// TIA Portal V20 export
// export: Created 2025-12-01T14:56:58.1690783Z, ExportSetting None, DisplayName Totally Integrated Automation Portal, DisplayVersion V20 Update 3, DisplayName TIA Portal Openness, DisplayVersion V20 Update 3, DisplayName TIA Portal Version Control Interface, DisplayVersion V20 Update 3, DisplayName STEP 7 Professional, DisplayVersion V20 Update 3, DisplayName STEP 7 Safety, DisplayVersion V20 Update 2, DisplayName WinCC Basic/Comfort/Advanced, DisplayVersion V20 Update 3, DisplayName WinCC Professional, DisplayVersion V20 Update 3, DisplayName WinCC Unified, DisplayVersion V20 Update 3
FUNCTION_BLOCK "FB86_GALIBO_3Laterales"   // FB86, LAD
TITLE = Galibo de 3 Anchuras (2024)
{ S7_Optimized_Access := 'FALSE' }
AUTHOR : GALIBO
NAME : 20140101
VERSION : 3.0
// stored: AutoNumber false, SetENOAutomatically false
   VAR_INPUT
      Mesa : UInt;
      NumGalibo : UInt;
      EnRodillos : Bool;
      pHs_Lateral_Dcha_Err : Bool;
      pHs_Lateral_Dcha_2 : Bool;
      pHs_Lateral_Dcha_1 : Bool;
      pHs_Lateral_Izq_1 : Bool;
      pHs_Lateral_Izq_2 : Bool;
      pHs_Lateral_Izq_Err : Bool;
      HabilitarLectura : Bool;
      PermisoLectura : Bool;
      Rearmar_ConMesaLibre : Bool;
   END_VAR
   VAR_OUTPUT
      Baliza : Bool;
      ErrorLateral : Bool;
      FinLectura : Bool;
   END_VAR
   VAR
      GAL_ET00 : Bool;
      GAL_ET01 : Bool;
      GAL_ET02 : Bool;
      GAL_ET03 : Bool;
      pHsGalibo_OK { ExternalAccessible := 'False'; ExternalVisible := 'False'; ExternalWritable := 'False'} : Bool;
      Lateral_NOOK_Dcha : Bool;
      Lateral_NOOK_Izq : Bool;
      Lateral_OK_1 : Bool;
      Lateral_OK_2 : Bool;
      Lateral_OK_3 : Bool;
      LeerLateral : Bool;
      CodigoLateral : SInt;
      MemoCodigo : Word;
      STAT_Baliza_Galibo : Bool;
   END_VAR
   VAR_TEMP
      EstadoZona : "EstadoZona";
      EstadoVI : "EstadosMesa";
   END_VAR
   VAR_TEMP   // added for the SCL form of the ladder/FBD networks
      _w1 : Bool;
   END_VAR
BEGIN

REGION Network 1: INICIALIZAR - Recoger las Variables de Estado de la Mesa
   // Se recoge - Estado_CBx
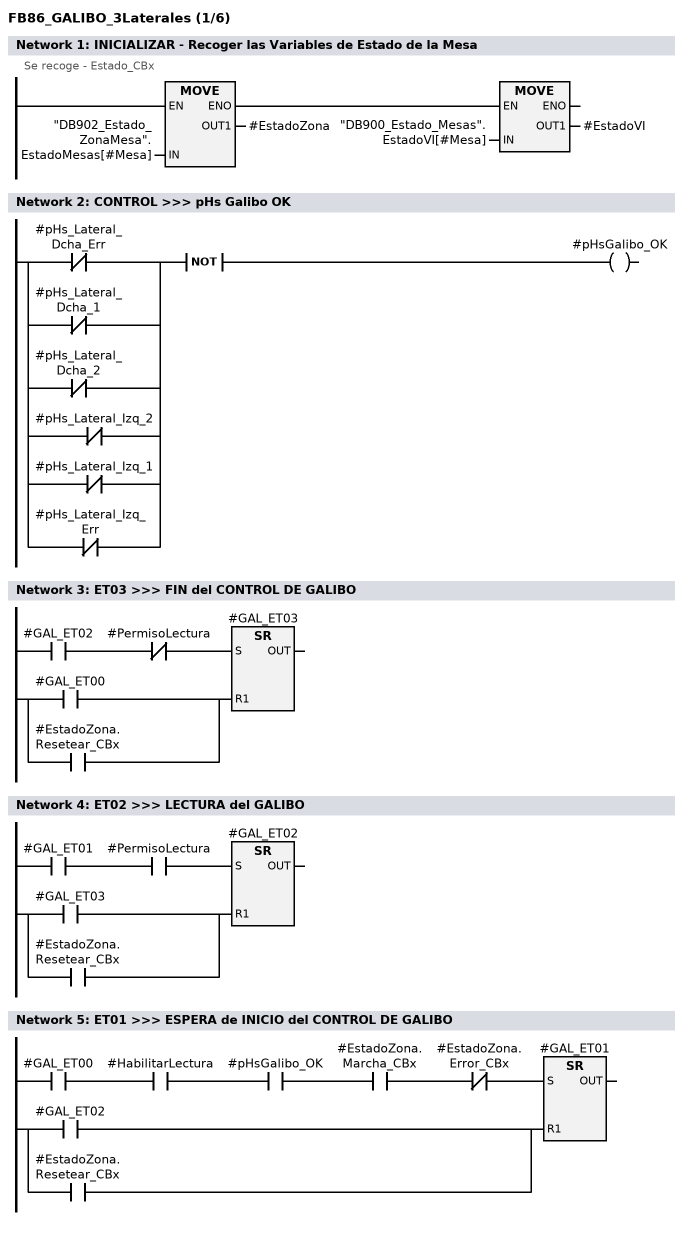
   RUNG wire#powerrail
      Move(in := "DB902_Estado_ZonaMesa".EstadoMesas[#Mesa], out1 => #EstadoZona)
      Move(in := "DB900_Estado_Mesas".EstadoVI[#Mesa], out1 => #EstadoVI)
   END_RUNG
   // the same network as SCL:
   #EstadoZona := "DB902_Estado_ZonaMesa".EstadoMesas[#Mesa];
   #EstadoVI := "DB900_Estado_Mesas".EstadoVI[#Mesa];
END_REGION

REGION Network 2: CONTROL >>> pHs Galibo OK
   RUNG wire#powerrail
      I_Contact( #pHs_Lateral_Dcha_Err )
      wire#w1
      Not()
      Coil( #pHsGalibo_OK )
   END_RUNG
   RUNG wire#powerrail
      I_Contact( #pHs_Lateral_Dcha_1 )
   END_RUNG wire#w1
   RUNG wire#powerrail
      I_Contact( #pHs_Lateral_Dcha_2 )
   END_RUNG wire#w1
   RUNG wire#powerrail
      I_Contact( #pHs_Lateral_Izq_2 )
   END_RUNG wire#w1
   RUNG wire#powerrail
      I_Contact( #pHs_Lateral_Izq_1 )
   END_RUNG wire#w1
   RUNG wire#powerrail
      I_Contact( #pHs_Lateral_Izq_Err )
   END_RUNG wire#w1
   // the same network as SCL:
   #pHsGalibo_OK := NOT (NOT #pHs_Lateral_Dcha_Err OR NOT #pHs_Lateral_Dcha_1 OR NOT #pHs_Lateral_Dcha_2 OR NOT #pHs_Lateral_Izq_2 OR NOT #pHs_Lateral_Izq_1 OR NOT #pHs_Lateral_Izq_Err);
END_REGION

REGION Network 3: ET03 >>> FIN del CONTROL DE GALIBO
   RUNG wire#powerrail
      Contact( #GAL_ET02 )
      I_Contact( #PermisoLectura )
      S_SR(operand := #GAL_ET03, r1 := wire#w1)
   END_RUNG
   RUNG wire#powerrail
      Contact( #GAL_ET00 )
   END_RUNG wire#w1
   RUNG wire#powerrail
      Contact( #EstadoZona.Resetear_CBx )
   END_RUNG wire#w1
   // the same network as SCL:
   IF #GAL_ET02 AND NOT #PermisoLectura THEN
       #GAL_ET03 := TRUE;   // SR flip-flop
   END_IF;
   IF #GAL_ET00 OR #EstadoZona.Resetear_CBx THEN #GAL_ET03 := FALSE; END_IF;
END_REGION

REGION Network 4: ET02 >>> LECTURA del GALIBO
   RUNG wire#powerrail
      Contact( #GAL_ET01 )
      Contact( #PermisoLectura )
      S_SR(operand := #GAL_ET02, r1 := wire#w1)
   END_RUNG
   RUNG wire#powerrail
      Contact( #GAL_ET03 )
   END_RUNG wire#w1
   RUNG wire#powerrail
      Contact( #EstadoZona.Resetear_CBx )
   END_RUNG wire#w1
   // the same network as SCL:
   IF #GAL_ET01 AND #PermisoLectura THEN
       #GAL_ET02 := TRUE;   // SR flip-flop
   END_IF;
   IF #GAL_ET03 OR #EstadoZona.Resetear_CBx THEN #GAL_ET02 := FALSE; END_IF;
END_REGION

REGION Network 5: ET01 >>> ESPERA de INICIO del CONTROL DE GALIBO
   RUNG wire#powerrail
      Contact( #GAL_ET00 )
      Contact( #HabilitarLectura )
      Contact( #pHsGalibo_OK )
      Contact( #EstadoZona.Marcha_CBx )
      I_Contact( #EstadoZona.Error_CBx )
      S_SR(operand := #GAL_ET01, r1 := wire#w1)
   END_RUNG
   RUNG wire#powerrail
      Contact( #GAL_ET02 )
   END_RUNG wire#w1
   RUNG wire#powerrail
      Contact( #EstadoZona.Resetear_CBx )
   END_RUNG wire#w1
   // the same network as SCL:
   IF #GAL_ET00 AND #HabilitarLectura AND #pHsGalibo_OK AND #EstadoZona.Marcha_CBx AND NOT #EstadoZona.Error_CBx THEN
       #GAL_ET01 := TRUE;   // SR flip-flop
   END_IF;
   IF #GAL_ET02 OR #EstadoZona.Resetear_CBx THEN #GAL_ET01 := FALSE; END_IF;
END_REGION

REGION Network 6: ET00 >>> INICIO
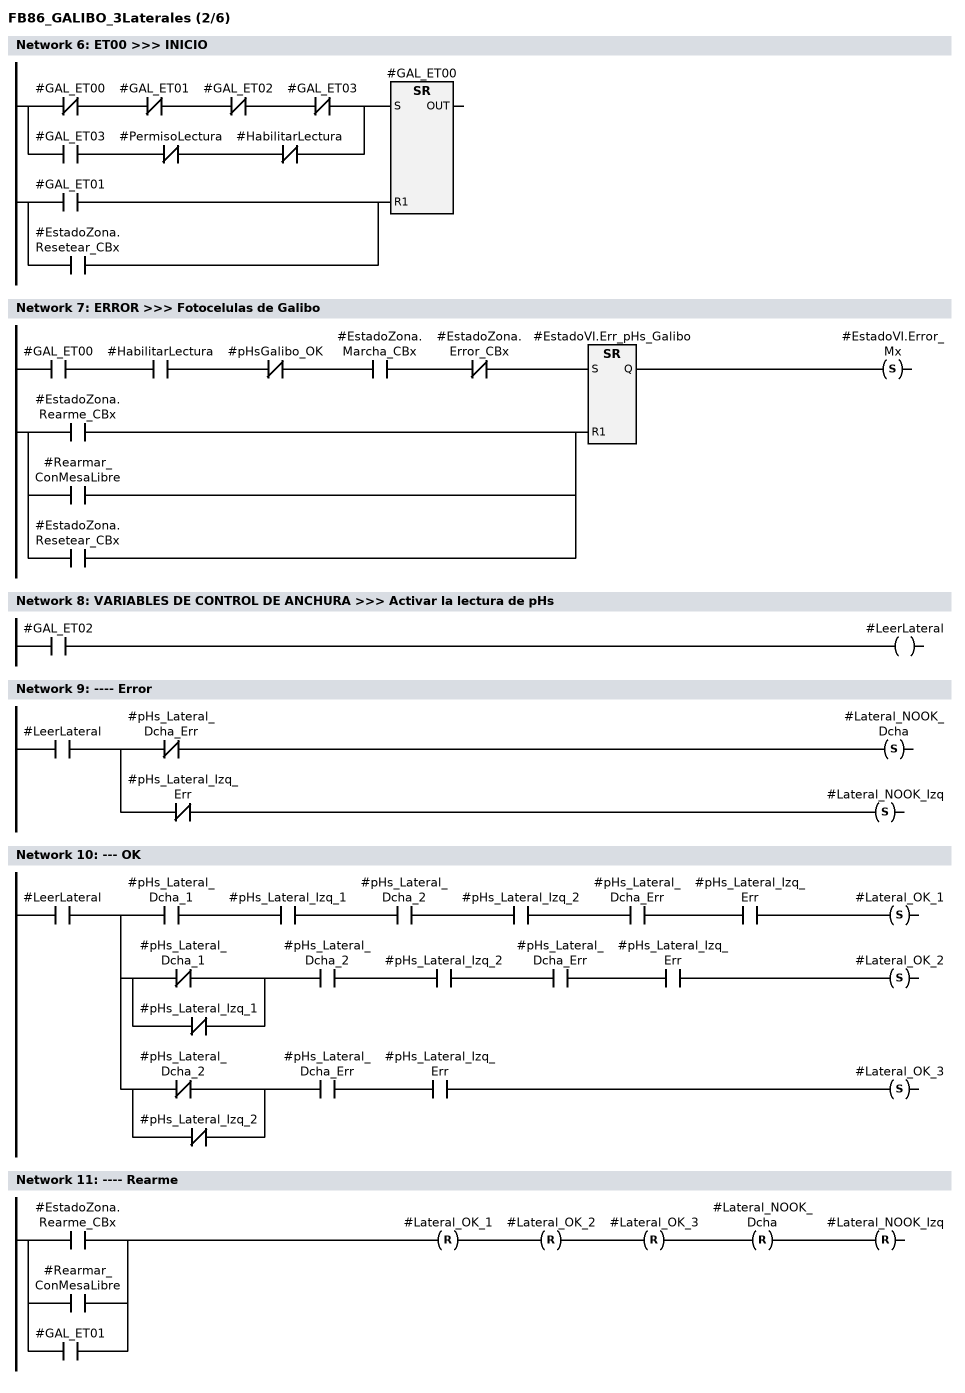
   RUNG wire#powerrail
      I_Contact( #GAL_ET00 )
      I_Contact( #GAL_ET01 )
      I_Contact( #GAL_ET02 )
      I_Contact( #GAL_ET03 )
      wire#w1
      S_SR(operand := #GAL_ET00, r1 := wire#w2)
   END_RUNG
   RUNG wire#powerrail
      Contact( #GAL_ET03 )
      I_Contact( #PermisoLectura )
      I_Contact( #HabilitarLectura )
   END_RUNG wire#w1
   RUNG wire#powerrail
      Contact( #GAL_ET01 )
   END_RUNG wire#w2
   RUNG wire#powerrail
      Contact( #EstadoZona.Resetear_CBx )
   END_RUNG wire#w2
   // the same network as SCL:
   IF (NOT #GAL_ET00 AND NOT #GAL_ET01 AND NOT #GAL_ET02 AND NOT #GAL_ET03) OR (#GAL_ET03 AND NOT #PermisoLectura AND NOT #HabilitarLectura) THEN
       #GAL_ET00 := TRUE;   // SR flip-flop
   END_IF;
   IF #GAL_ET01 OR #EstadoZona.Resetear_CBx THEN #GAL_ET00 := FALSE; END_IF;
END_REGION

REGION Network 7: ERROR >>> Fotocelulas de Galibo
   RUNG wire#powerrail
      Contact( #GAL_ET00 )
      Contact( #HabilitarLectura )
      I_Contact( #pHsGalibo_OK )
      Contact( #EstadoZona.Marcha_CBx )
      I_Contact( #EstadoZona.Error_CBx )
      S_SR(operand := #EstadoVI.Err_pHs_Galibo, r1 := wire#w1)
      S_Coil( #EstadoVI.Error_Mx )
   END_RUNG
   RUNG wire#powerrail
      Contact( #EstadoZona.Rearme_CBx )
   END_RUNG wire#w1
   RUNG wire#powerrail
      Contact( #Rearmar_ConMesaLibre )
   END_RUNG wire#w1
   RUNG wire#powerrail
      Contact( #EstadoZona.Resetear_CBx )
   END_RUNG wire#w1
   // the same network as SCL:
   IF #GAL_ET00 AND #HabilitarLectura AND NOT #pHsGalibo_OK AND #EstadoZona.Marcha_CBx AND NOT #EstadoZona.Error_CBx THEN
       #EstadoVI.Err_pHs_Galibo := TRUE;   // SR flip-flop
   END_IF;
   IF #EstadoZona.Rearme_CBx OR #Rearmar_ConMesaLibre OR #EstadoZona.Resetear_CBx THEN
       #EstadoVI.Err_pHs_Galibo := FALSE;
   END_IF;
   IF #EstadoVI.Err_pHs_Galibo THEN #EstadoVI.Error_Mx := TRUE; END_IF;
END_REGION

REGION Network 8: VARIABLES DE CONTROL DE ANCHURA >>> Activar la lectura de pHs
   RUNG wire#powerrail
      Contact( #GAL_ET02 )
      Coil( #LeerLateral )
   END_RUNG
   // the same network as SCL:
   #LeerLateral := #GAL_ET02;
END_REGION

REGION Network 9: ---- Error
   RUNG wire#powerrail
      Contact( #LeerLateral )
      wire#w1
      I_Contact( #pHs_Lateral_Dcha_Err )
      S_Coil( #Lateral_NOOK_Dcha )
   END_RUNG
   RUNG wire#w1
      I_Contact( #pHs_Lateral_Izq_Err )
      S_Coil( #Lateral_NOOK_Izq )
   END_RUNG
   // the same network as SCL:
   IF #LeerLateral AND NOT #pHs_Lateral_Dcha_Err THEN #Lateral_NOOK_Dcha := TRUE; END_IF;
   IF #LeerLateral AND NOT #pHs_Lateral_Izq_Err THEN #Lateral_NOOK_Izq := TRUE; END_IF;
END_REGION

REGION Network 10: --- OK
   RUNG wire#powerrail
      Contact( #LeerLateral )
      wire#w1
      Contact( #pHs_Lateral_Dcha_1 )
      Contact( #pHs_Lateral_Izq_1 )
      Contact( #pHs_Lateral_Dcha_2 )
      Contact( #pHs_Lateral_Izq_2 )
      Contact( #pHs_Lateral_Dcha_Err )
      Contact( #pHs_Lateral_Izq_Err )
      S_Coil( #Lateral_OK_1 )
   END_RUNG
   RUNG wire#w1
      I_Contact( #pHs_Lateral_Dcha_1 )
      wire#w2
      Contact( #pHs_Lateral_Dcha_2 )
      Contact( #pHs_Lateral_Izq_2 )
      Contact( #pHs_Lateral_Dcha_Err )
      Contact( #pHs_Lateral_Izq_Err )
      S_Coil( #Lateral_OK_2 )
   END_RUNG
   RUNG wire#w1
      I_Contact( #pHs_Lateral_Izq_1 )
   END_RUNG wire#w2
   RUNG wire#w1
      I_Contact( #pHs_Lateral_Dcha_2 )
      wire#w3
      Contact( #pHs_Lateral_Dcha_Err )
      Contact( #pHs_Lateral_Izq_Err )
      S_Coil( #Lateral_OK_3 )
   END_RUNG
   RUNG wire#w1
      I_Contact( #pHs_Lateral_Izq_2 )
   END_RUNG wire#w3
   // the same network as SCL:
   IF #LeerLateral AND #pHs_Lateral_Dcha_1 AND #pHs_Lateral_Izq_1 AND #pHs_Lateral_Dcha_2 AND #pHs_Lateral_Izq_2 AND #pHs_Lateral_Dcha_Err AND #pHs_Lateral_Izq_Err THEN
       #Lateral_OK_1 := TRUE;
   END_IF;
   IF #LeerLateral AND (NOT #pHs_Lateral_Dcha_1 OR NOT #pHs_Lateral_Izq_1) AND #pHs_Lateral_Dcha_2 AND #pHs_Lateral_Izq_2 AND #pHs_Lateral_Dcha_Err AND #pHs_Lateral_Izq_Err THEN
       #Lateral_OK_2 := TRUE;
   END_IF;
   IF #LeerLateral AND (NOT #pHs_Lateral_Dcha_2 OR NOT #pHs_Lateral_Izq_2) AND #pHs_Lateral_Dcha_Err AND #pHs_Lateral_Izq_Err THEN
       #Lateral_OK_3 := TRUE;
   END_IF;
END_REGION

REGION Network 11: ---- Rearme
   RUNG wire#powerrail
      Contact( #EstadoZona.Rearme_CBx )
      wire#w1
      R_Coil( #Lateral_OK_1 )
      R_Coil( #Lateral_OK_2 )
      R_Coil( #Lateral_OK_3 )
      R_Coil( #Lateral_NOOK_Dcha )
      R_Coil( #Lateral_NOOK_Izq )
   END_RUNG
   RUNG wire#powerrail
      Contact( #Rearmar_ConMesaLibre )
   END_RUNG wire#w1
   RUNG wire#powerrail
      Contact( #GAL_ET01 )
   END_RUNG wire#w1
   // the same network as SCL:
   IF #EstadoZona.Rearme_CBx OR #Rearmar_ConMesaLibre OR #GAL_ET01 THEN
       #Lateral_OK_1 := FALSE;
       #Lateral_OK_2 := FALSE;
       #Lateral_OK_3 := FALSE;
       #Lateral_NOOK_Dcha := FALSE;
       #Lateral_NOOK_Izq := FALSE;
   END_IF;
END_REGION

REGION Network 12: CODIFICACION DEL GALIBO >>> Inicialiar
   // Por Defecto >>> Sin realizar lectura
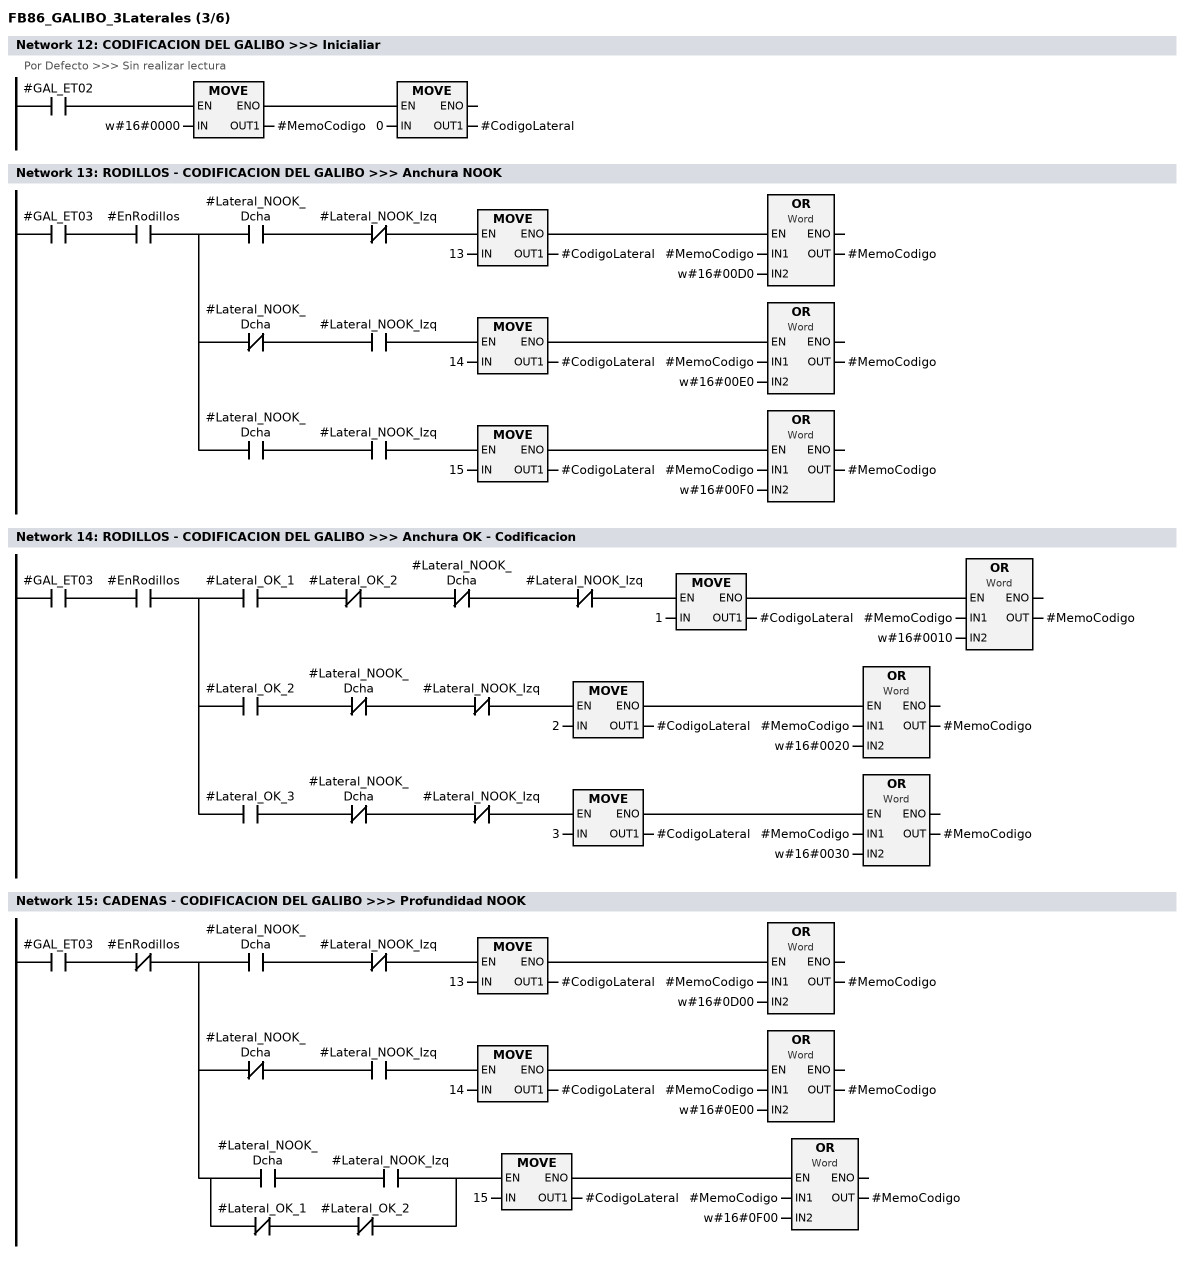
   RUNG wire#powerrail
      Contact( #GAL_ET02 )
      { S7_GenerateENO := "TRUE" } Move(in := w#16#0000, out1 => #MemoCodigo)
      { S7_GenerateENO := "TRUE" } Move(in := 0, out1 => #CodigoLateral)
   END_RUNG
   // the same network as SCL:
   // ENO of a box is taken as its EN; it also drops when the box reports an error
   IF #GAL_ET02 THEN
       #MemoCodigo := w#16#0000;
       #CodigoLateral := 0;
   END_IF;
END_REGION

REGION Network 13: RODILLOS - CODIFICACION DEL GALIBO >>> Anchura NOOK
   #_w1 := #GAL_ET03 AND #EnRodillos;
   IF #_w1 AND #Lateral_NOOK_Dcha AND NOT #Lateral_NOOK_Izq THEN
       #CodigoLateral := 13;
       #MemoCodigo := #MemoCodigo OR w#16#00D0;
   END_IF;
   IF #_w1 AND NOT #Lateral_NOOK_Dcha AND #Lateral_NOOK_Izq THEN
       #CodigoLateral := 14;
       #MemoCodigo := #MemoCodigo OR w#16#00E0;
   END_IF;
   IF #_w1 AND #Lateral_NOOK_Dcha AND #Lateral_NOOK_Izq THEN
       #CodigoLateral := 15;
       #MemoCodigo := #MemoCodigo OR w#16#00F0;
   END_IF;
END_REGION

REGION Network 14: RODILLOS - CODIFICACION DEL GALIBO >>> Anchura OK - Codificacion
   #_w1 := #GAL_ET03 AND #EnRodillos;
   IF #_w1 AND #Lateral_OK_1 AND NOT #Lateral_OK_2 AND NOT #Lateral_NOOK_Dcha AND NOT #Lateral_NOOK_Izq THEN
       #CodigoLateral := 1;
       #MemoCodigo := #MemoCodigo OR w#16#0010;
   END_IF;
   IF #_w1 AND #Lateral_OK_2 AND NOT #Lateral_NOOK_Dcha AND NOT #Lateral_NOOK_Izq THEN
       #CodigoLateral := 2;
       #MemoCodigo := #MemoCodigo OR w#16#0020;
   END_IF;
   IF #_w1 AND #Lateral_OK_3 AND NOT #Lateral_NOOK_Dcha AND NOT #Lateral_NOOK_Izq THEN
       #CodigoLateral := 3;
       #MemoCodigo := #MemoCodigo OR w#16#0030;
   END_IF;
END_REGION

REGION Network 15: CADENAS - CODIFICACION DEL GALIBO >>> Profundidad NOOK
   #_w1 := #GAL_ET03 AND NOT #EnRodillos;
   IF #_w1 AND #Lateral_NOOK_Dcha AND NOT #Lateral_NOOK_Izq THEN
       #CodigoLateral := 13;
       #MemoCodigo := #MemoCodigo OR w#16#0D00;
   END_IF;
   IF #_w1 AND NOT #Lateral_NOOK_Dcha AND #Lateral_NOOK_Izq THEN
       #CodigoLateral := 14;
       #MemoCodigo := #MemoCodigo OR w#16#0E00;
   END_IF;
   IF #_w1 AND ((#Lateral_NOOK_Dcha AND #Lateral_NOOK_Izq) OR (NOT #Lateral_OK_1 AND NOT #Lateral_OK_2)) THEN
       #CodigoLateral := 15;
       #MemoCodigo := #MemoCodigo OR w#16#0F00;
   END_IF;
END_REGION

REGION Network 16: CADENAS - CODIFICACION DEL GALIBO >>> Profundidad OK - Codificacion
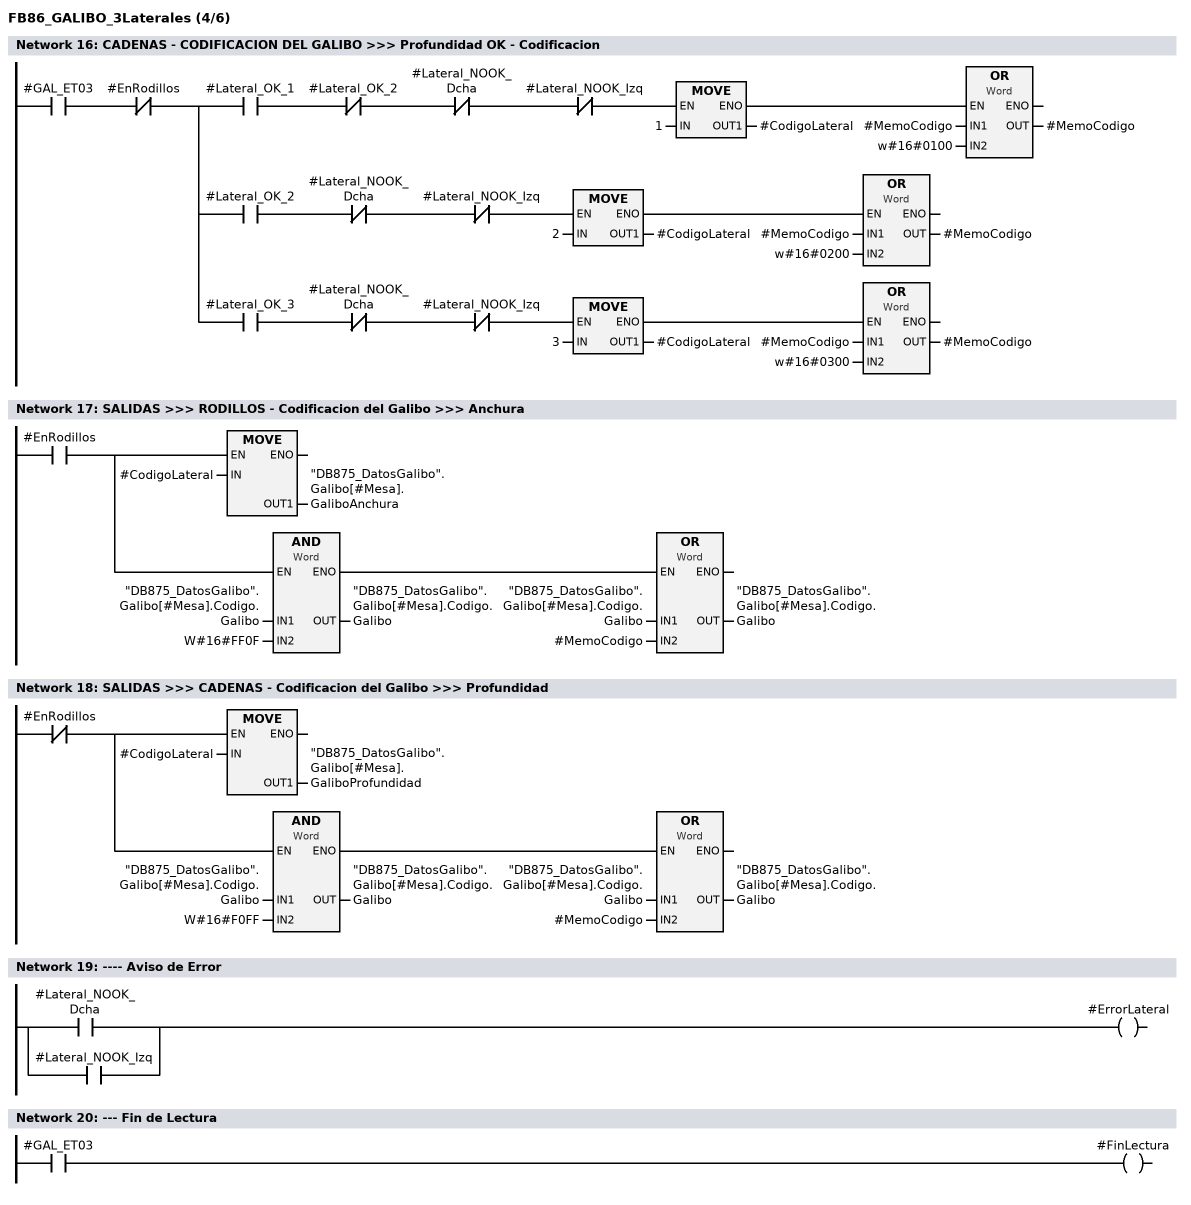
   #_w1 := #GAL_ET03 AND NOT #EnRodillos;
   IF #_w1 AND #Lateral_OK_1 AND NOT #Lateral_OK_2 AND NOT #Lateral_NOOK_Dcha AND NOT #Lateral_NOOK_Izq THEN
       #CodigoLateral := 1;
       #MemoCodigo := #MemoCodigo OR w#16#0100;
   END_IF;
   IF #_w1 AND #Lateral_OK_2 AND NOT #Lateral_NOOK_Dcha AND NOT #Lateral_NOOK_Izq THEN
       #CodigoLateral := 2;
       #MemoCodigo := #MemoCodigo OR w#16#0200;
   END_IF;
   IF #_w1 AND #Lateral_OK_3 AND NOT #Lateral_NOOK_Dcha AND NOT #Lateral_NOOK_Izq THEN
       #CodigoLateral := 3;
       #MemoCodigo := #MemoCodigo OR w#16#0300;
   END_IF;
END_REGION

REGION Network 17: SALIDAS >>> RODILLOS - Codificacion del Galibo >>> Anchura
   IF #EnRodillos THEN
       "DB875_DatosGalibo".Galibo[#Mesa].GaliboAnchura := #CodigoLateral;
       "DB875_DatosGalibo".Galibo[#Mesa].Codigo.Galibo := "DB875_DatosGalibo".Galibo[#Mesa].Codigo.Galibo AND W#16#FF0F;
       "DB875_DatosGalibo".Galibo[#Mesa].Codigo.Galibo := "DB875_DatosGalibo".Galibo[#Mesa].Codigo.Galibo OR #MemoCodigo;
   END_IF;
END_REGION

REGION Network 18: SALIDAS >>> CADENAS - Codificacion del Galibo >>> Profundidad
   IF NOT #EnRodillos THEN
       "DB875_DatosGalibo".Galibo[#Mesa].GaliboProfundidad := #CodigoLateral;
       "DB875_DatosGalibo".Galibo[#Mesa].Codigo.Galibo := "DB875_DatosGalibo".Galibo[#Mesa].Codigo.Galibo AND W#16#F0FF;
       "DB875_DatosGalibo".Galibo[#Mesa].Codigo.Galibo := "DB875_DatosGalibo".Galibo[#Mesa].Codigo.Galibo OR #MemoCodigo;
   END_IF;
END_REGION

REGION Network 19: ---- Aviso de Error
   RUNG wire#powerrail
      Contact( #Lateral_NOOK_Dcha )
      wire#w1
      Coil( #ErrorLateral )
   END_RUNG
   RUNG wire#powerrail
      Contact( #Lateral_NOOK_Izq )
   END_RUNG wire#w1
   // the same network as SCL:
   #ErrorLateral := #Lateral_NOOK_Dcha OR #Lateral_NOOK_Izq;
END_REGION

REGION Network 20: --- Fin de Lectura
   RUNG wire#powerrail
      Contact( #GAL_ET03 )
      Coil( #FinLectura )
   END_RUNG
   // the same network as SCL:
   #FinLectura := #GAL_ET03;
END_REGION

REGION Network 21: SALIDAS >>> BALIZA
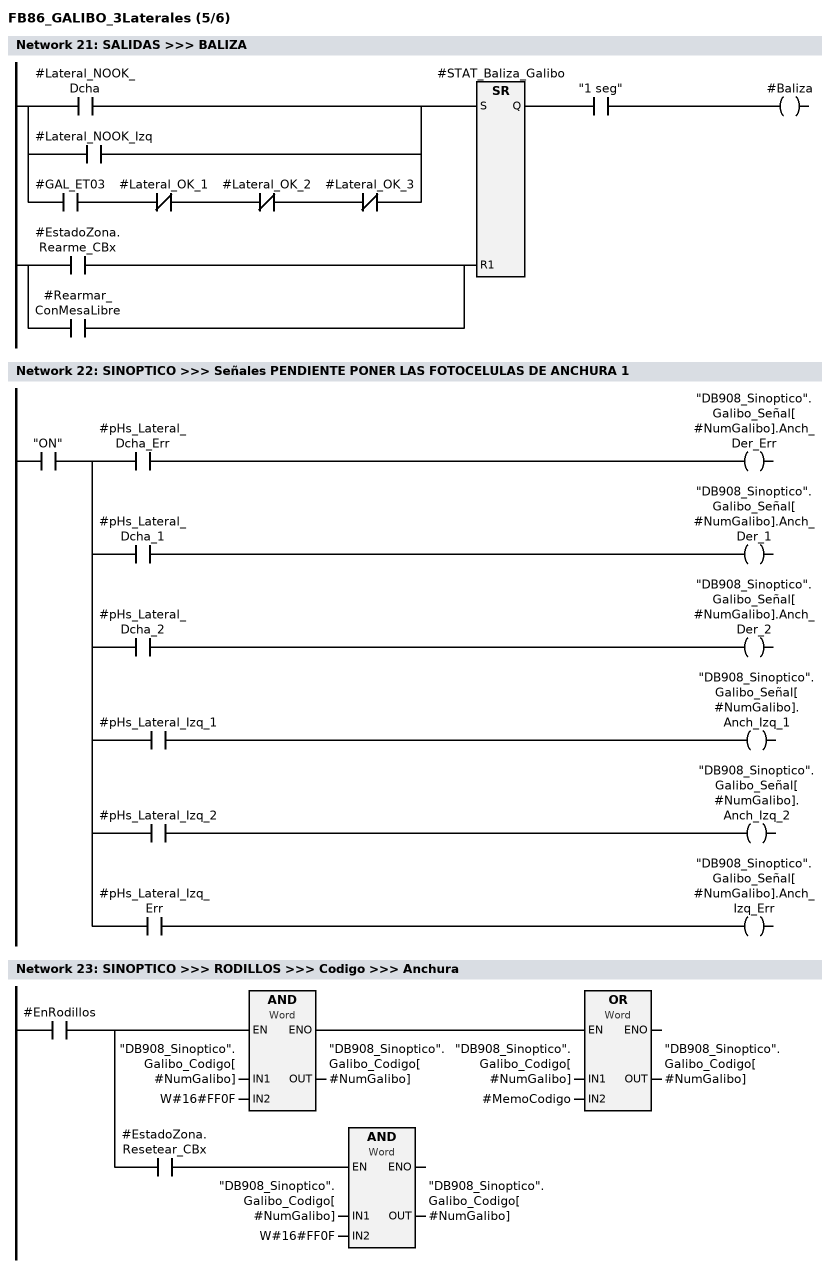
   RUNG wire#powerrail
      Contact( #Lateral_NOOK_Dcha )
      wire#w1
      S_SR(operand := #STAT_Baliza_Galibo, r1 := wire#w2)
      Contact( "1 seg" )
      Coil( #Baliza )
   END_RUNG
   RUNG wire#powerrail
      Contact( #Lateral_NOOK_Izq )
   END_RUNG wire#w1
   RUNG wire#powerrail
      Contact( #GAL_ET03 )
      I_Contact( #Lateral_OK_1 )
      I_Contact( #Lateral_OK_2 )
      I_Contact( #Lateral_OK_3 )
   END_RUNG wire#w1
   RUNG wire#powerrail
      Contact( #EstadoZona.Rearme_CBx )
   END_RUNG wire#w2
   RUNG wire#powerrail
      Contact( #Rearmar_ConMesaLibre )
   END_RUNG wire#w2
   // the same network as SCL:
   IF #Lateral_NOOK_Dcha OR #Lateral_NOOK_Izq OR (#GAL_ET03 AND NOT #Lateral_OK_1 AND NOT #Lateral_OK_2 AND NOT #Lateral_OK_3) THEN
       #STAT_Baliza_Galibo := TRUE;   // SR flip-flop
   END_IF;
   IF #EstadoZona.Rearme_CBx OR #Rearmar_ConMesaLibre THEN #STAT_Baliza_Galibo := FALSE; END_IF;
   #Baliza := #STAT_Baliza_Galibo AND "1 seg";
END_REGION

REGION Network 22: SINOPTICO >>> Señales PENDIENTE PONER LAS FOTOCELULAS DE ANCHURA 1
   RUNG wire#powerrail
      Contact( "ON" )
      wire#w1
      Contact( #pHs_Lateral_Dcha_Err )
      Coil( "DB908_Sinoptico".Galibo_Señal[#NumGalibo].Anch_Der_Err )
   END_RUNG
   RUNG wire#w1
      Contact( #pHs_Lateral_Dcha_1 )
      Coil( "DB908_Sinoptico".Galibo_Señal[#NumGalibo].Anch_Der_1 )
   END_RUNG
   RUNG wire#w1
      Contact( #pHs_Lateral_Dcha_2 )
      Coil( "DB908_Sinoptico".Galibo_Señal[#NumGalibo].Anch_Der_2 )
   END_RUNG
   RUNG wire#w1
      Contact( #pHs_Lateral_Izq_1 )
      Coil( "DB908_Sinoptico".Galibo_Señal[#NumGalibo].Anch_Izq_1 )
   END_RUNG
   RUNG wire#w1
      Contact( #pHs_Lateral_Izq_2 )
      Coil( "DB908_Sinoptico".Galibo_Señal[#NumGalibo].Anch_Izq_2 )
   END_RUNG
   RUNG wire#w1
      Contact( #pHs_Lateral_Izq_Err )
      Coil( "DB908_Sinoptico".Galibo_Señal[#NumGalibo].Anch_Izq_Err )
   END_RUNG
   // the same network as SCL:
   "DB908_Sinoptico".Galibo_Señal[#NumGalibo].Anch_Der_Err := "ON" AND #pHs_Lateral_Dcha_Err;
   "DB908_Sinoptico".Galibo_Señal[#NumGalibo].Anch_Der_1 := "ON" AND #pHs_Lateral_Dcha_1;
   "DB908_Sinoptico".Galibo_Señal[#NumGalibo].Anch_Der_2 := "ON" AND #pHs_Lateral_Dcha_2;
   "DB908_Sinoptico".Galibo_Señal[#NumGalibo].Anch_Izq_1 := "ON" AND #pHs_Lateral_Izq_1;
   "DB908_Sinoptico".Galibo_Señal[#NumGalibo].Anch_Izq_2 := "ON" AND #pHs_Lateral_Izq_2;
   "DB908_Sinoptico".Galibo_Señal[#NumGalibo].Anch_Izq_Err := "ON" AND #pHs_Lateral_Izq_Err;
END_REGION

REGION Network 23: SINOPTICO >>> RODILLOS >>> Codigo >>> Anchura
   IF #EnRodillos THEN
       "DB908_Sinoptico".Galibo_Codigo[#NumGalibo] := "DB908_Sinoptico".Galibo_Codigo[#NumGalibo] AND W#16#FF0F;
       "DB908_Sinoptico".Galibo_Codigo[#NumGalibo] := "DB908_Sinoptico".Galibo_Codigo[#NumGalibo] OR #MemoCodigo;
   END_IF;
   IF #EnRodillos AND #EstadoZona.Resetear_CBx THEN
       "DB908_Sinoptico".Galibo_Codigo[#NumGalibo] := "DB908_Sinoptico".Galibo_Codigo[#NumGalibo] AND W#16#FF0F;
   END_IF;
END_REGION

REGION Network 24: SINOPTICO >>> CADENAS >>> Codigo >>> Profundidad
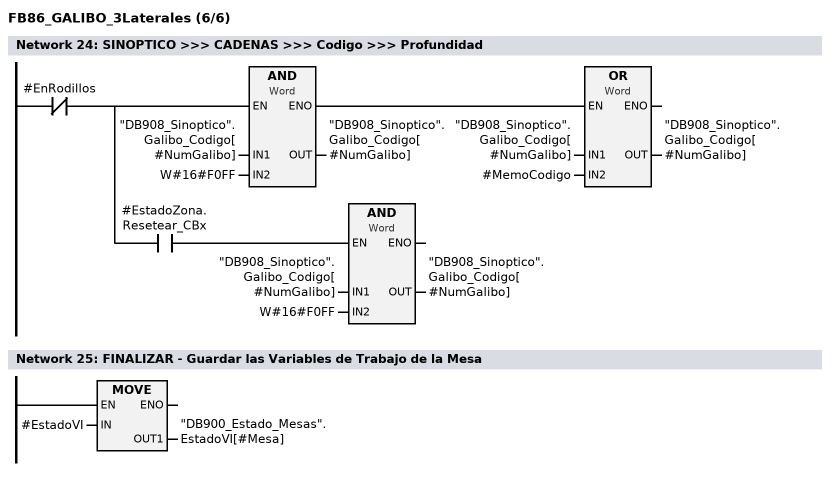
   IF NOT #EnRodillos THEN
       "DB908_Sinoptico".Galibo_Codigo[#NumGalibo] := "DB908_Sinoptico".Galibo_Codigo[#NumGalibo] AND W#16#F0FF;
       "DB908_Sinoptico".Galibo_Codigo[#NumGalibo] := "DB908_Sinoptico".Galibo_Codigo[#NumGalibo] OR #MemoCodigo;
   END_IF;
   IF NOT #EnRodillos AND #EstadoZona.Resetear_CBx THEN
       "DB908_Sinoptico".Galibo_Codigo[#NumGalibo] := "DB908_Sinoptico".Galibo_Codigo[#NumGalibo] AND W#16#F0FF;
   END_IF;
END_REGION

REGION Network 25: FINALIZAR - Guardar las Variables de Trabajo de la Mesa
   RUNG wire#powerrail
      Move(in := #EstadoVI, out1 => "DB900_Estado_Mesas".EstadoVI[#Mesa])
   END_RUNG
   // the same network as SCL:
   "DB900_Estado_Mesas".EstadoVI[#Mesa] := #EstadoVI;
END_REGION
END_FUNCTION_BLOCK
